FUNCTION TryConvert_WORD_TO_WORD : BOOL
VAR_INPUT
	in : WORD;
	out : REFERENCE TO WORD;
END_VAR

out := in;
TryConvert_WORD_TO_WORD := TRUE;

END_FUNCTION

(* stored: Version 1.1.0.1, ProductVersion 3.1.4024.12
   POU TryConvert_WORD_TO_WORD: Id {1c15fe9b-bb48-4a61-928a-d7d0d8ffdf04}, SpecialFunc None *)
